FUNCTION_BLOCK Basic (* Basic Function Block Type *)
  (* Standard: 61499-2 *)
  (* Version 0.2, 2003-12-04, JHC, Rockwell Automation, Renamed for better indexing. *)
  (* Version 0.1, 2002-11-05, JHC, Rockwell Automation, Corrected missing ST element in Algorithm REQ. *)
  (* Version 0.0, 2000-05-30, JHC, Rockwell Automation *)
  (* Compiler header: package fb.rt.cs725; *)
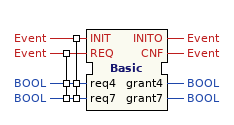
  EVENT_INPUT
    INIT WITH req4, req7; (* Initialization Request *)
    REQ WITH req4, req7; (* Normal Execution Request *)
  END_EVENT
  EVENT_OUTPUT
    INITO; (* Initialization Confirm *)
    CNF; (* Execution Confirmation *)
  END_EVENT
  VAR_INPUT
    req4 : BOOL; (* Input event qualifier *)
    req7 : BOOL;
  END_VAR
  VAR_OUTPUT
    grant4 : BOOL;
    grant7 : BOOL;
  END_VAR
  VAR
    requests : ARRAY [0..1] OF ARRAY;
  END_VAR
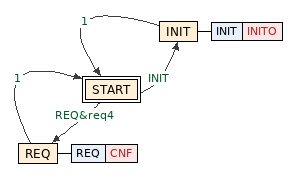
  EC_STATES
    START; (* Initial State *)
    INIT : INIT -> INITO; (* Initialization *)
    REQ : REQ -> CNF; (* Normal execution *)
  END_STATES
  EC_TRANSITIONS
    START TO INIT := INIT;
    INIT TO START := 1;
    START TO REQ := REQ&req4;
    REQ TO START := 1;
  END_TRANSITIONS
  ALGORITHM INIT IN Java: (* Initialization algorithm *)
grant4.value=false;
grant7.value=false;
requests[0] = 0;
requests[1] = 0;
  END_ALGORITHM
  ALGORITHM REQ IN Java: (* Normally executed algorithm *)
int requests[];
  END_ALGORITHM
END_FUNCTION_BLOCK
